// TwinCAT 3 PLC project Soft_PLC
// ProgramVersion: 3.1.4024.0
// libraries:
//   Tc2_Standard, * (Beckhoff Automation GmbH)
//   Tc2_System, * (Beckhoff Automation GmbH)
//   Tc3_Module, * (Beckhoff Automation GmbH)
// project tree:
//   / PlcTask.TcTTO
//   POUs/ MAIN.TcPOU
// real-time tasks:
//   TASK PlcTask: cycle T#10ms, priority 20, ADS port 350

CONFIGURATION Soft_PLC
    RESOURCE PLC ON TwinCAT3
        TASK PlcTask(INTERVAL := T#10ms, PRIORITY := 20);
        PROGRAM MAIN WITH PlcTask : MAIN;
    END_RESOURCE
END_CONFIGURATION

// ---- POUs/MAIN.TcPOU
PROGRAM MAIN
VAR
	bRun_Process : BOOL;
	bStop_process : BOOL;
	bProcess_Status : BOOL;
	tProcess_Duration : TIME;
	fbProcess_Timer : TON;
	bTimer_Done : BOOL;	
END_VAR

//bProcess_Status := bRun_Process;

fbProcess_Timer(IN:= bProcess_Status, PT:= tProcess_Duration, Q=> bTimer_Done, ET=> );


IF bRun_Process THEN
	bProcess_Status := TRUE;
END_IF

IF bStop_Process OR bTimer_Done THEN
	bProcess_Status := FALSE;
END_IF

END_PROGRAM
